{attribute addProperty BoxType "EL3783-0000-0018"}
{attribute addProperty Id "U1_SamplesAT %I*ARRAY [0..19] OF INT32040"}
{attribute addProperty CRC "1704852166"}
{attribute addProperty SizeInBites "320"}
{attribute addProperty SizeInBytes "40"}
TYPE L1_Voltage_Samples_659DFAC6 :
STRUCT
	{attribute addProperty Name "U1_Samples"}
	U1_Samples AT %I* : ARRAY [0..19] OF INT;
END_STRUCT
END_TYPE

(* stored: Version 1.2.0.0, ProductVersion 3.1.4024.9
   DUT L1_Voltage_Samples_659DFAC6: Id {bfcff8e3-1bb6-49da-b2c0-25dc16007c05} *)
